Staubli VAL3: setCycle.pgx

public program setCycle(string x_sName, num x_nTotal, num x_nDone, num x_nIndex, num x_nType)
begin
  // insert one cycle in the processLIST
  switch x_nType
    case 0
      // ON START CYCLE
      logMsg("[KERNEL] CYCLE:Insert the program: "+x_sName+" at the position: "+toString("",x_nIndex))
      saveCycle:sLoadStart[x_nIndex]=x_sName
      saveCycle:nTotalStart[x_nIndex]=x_nTotal
      saveCycle:nDoneStart[x_nIndex]=x_nDone
    break
    case 1
      // get the information about the actual process list
      logMsg("[KERNEL] CYCLE:Insert the program: "+x_sName+" at the position: "+toString("",x_nIndex))
      saveCycle:sLoadProg[x_nIndex]=x_sName
      saveCycle:nTotalCycle[x_nIndex]=x_nTotal
      saveCycle:nDoneCycle[x_nIndex]=x_nDone
    break
    case 2
      // ON END CYCLE
      logMsg("[KERNEL] CYCLE:Insert the program: "+x_sName+" at the position: "+toString("",x_nIndex))
      saveCycle:sLoadEnd[x_nIndex]=x_sName
      saveCycle:nTotalEnd[x_nIndex]=x_nTotal
      saveCycle:nDoneEnd[x_nIndex]=x_nDone
    break
  endSwitch
end
